TYPE ST_EL2809_A :
STRUCT
	//--------------------------------------------------------------------------------------------------------
	sTerminalName                                           :   STRING(200):= 'EL2809 | 16-Channel Digital Output';
	//=============================================================================================================
	// TERMINAL - EL2809	16-Channel Digital Output Terminal	 (Term 9)
	qStartButtonLED							AT %Q*			: 	BOOL;	// EL2809 channel 1
	qResetButtonLED							AT %Q* 			: 	BOOL;	// EL2809 channel 2
	qOpenProcessDoor             			AT %Q*	 		: 	BOOL;	// EL2809 channel 3 			
	qCloseProcessDoor      					AT %Q*	 		: 	BOOL;	// EL2809 channel 4 
	qExtendProcessCylinder1			  		AT %Q*	 		: 	BOOL;	// EL2809 channel 5
	qRetractProcessCylinder1			 	AT %Q*	 		: 	BOOL;	// EL2809 channel 6 	
	qPanelLightLED         		    		AT %Q*			: 	BOOL;	// EL2809 channel 7	
	qIndicatorLED1_Red						AT %Q*	 		: 	BOOL;	// EL2809 channel 8	
	qIndicatorLED1_Green                 	AT %Q*          :   BOOL;   // EL2809 channel 9
	qIndicatorLED2_Red             			AT %Q*          :   BOOL;   // EL2809 channel 10   	
	qIndicatorLED2_Green     				AT %Q*	 		: 	BOOL;	// EL2809 channel 11	
	qPartHolder1 							AT %Q*	 		: 	BOOL;	// EL2809 channel 12 
    iEL2809_A_Ch13							AT %Q*	 		: 	BOOL;	// EL2809 channel 13 
	qExtendVacuumCylinder1                	AT %Q*	 		: 	BOOL;	// EL2809 channel 14 
	qRetractVacuumCylinder1					AT %Q*	 		: 	BOOL;	// EL2809 channel 15 
    qPuckLockerPinCommand  	        		AT %Q*	 		: 	BOOL;	// EL2809 channel 16
	
	stTerminalInfo											: 	ST_Terminal_Info;

END_STRUCT
END_TYPE

(* stored: Version 1.1.0.1, ProductVersion 3.1.4026.18
   DUT ST_EL2809_A: Id {b4247617-0c63-4291-9ee1-02e0a92b28da} *)
